TYPE E_CoatingPosition :
(
    COA_Upper := 0,
    COA_Lower := 1,
    COA_Unknown := 2
) INT;
END_TYPE

(* stored: Version 1.1.0.1, ProductVersion 3.1.4024.12
   DUT E_CoatingPosition: Id {14085036-a3de-4738-a5ff-6c770eed6f44} *)
